// TIA Portal V20 export
DATA_BLOCK "Instance_FB_Start_Test_DB"   // DB105
// stored: AutoNumber false, InstanceOfName FB_Start_Test, InstanceOfType FB
"FB_Start_Test"
   // VAR_INPUT
   //    Button_Start_Approve : Bool;
   //    Electrical_Current_Test_Approved : Bool;
   //    Visual_Test_Approved_PLC : Bool;
   //    Reset_Funcional_Test : Bool;
   // END_VAR
   // VAR_OUTPUT
   //    Start_Functional_Test : Bool;
   //    Blink_Button_Light : Bool;
   //    Turn_On_Button_Light : Bool;
   //    Light_Fail_Test : Bool;
   //    Light_Approve_Test : Bool;
   // END_VAR
   // VAR
   //    Aux_Trigger_0 : Bool;
   // END_VAR
BEGIN
END_DATA_BLOCK
